VAR_GLOBAL
    // Arbiter linked to the FFO and the MPS
//    {attribute 'pytmc' := 'pv: PLC:TMO:MOTION:ARB'}
    fbArbiter: FB_Arbiter(1);

    // Fast fault for before ST4K4 (Most Devices)
//    {attribute 'pytmc' := 'pv: PLC:TMO:MOTION:FFO:01'}
//    {attribute 'TcLinkTo' := '.q_xFastFaultOut:=TIIB[PMPS_FFO]^Channel 1^Output'}
    fbFastFaultOutput1: FB_HardwareFFOutput := (bAutoReset := TRUE, i_sNetID:='172.21.92.73.1.1');
    // Fast fault for after ST4K4 (Basically just DREAM)
//    {attribute 'pytmc' := 'pv: PLC:TMO:MOTION:FFO:02'}
//    {attribute 'TcLinkTo' := '.q_xFastFaultOut:=TIIB[PMPS_FFO]^Channel 2^Output'}
//    fbFastFaultOutput2: FB_HardwareFFOutput := (bAutoReset := TRUE, i_sNetID:='172.21.92.73.1.1');
END_VAR

(* stored: Version 1.1.0.1, ProductVersion 3.1.4024.6
   GVL PMPS: Id {a2bc0a56-5468-49fb-a679-7c59628f5fcd} *)
